PROGRAM P50_RecipeControl1
VAR
	RcpIndex	: INT;
	
	iTimerCount: INT;
	OnTimer: TON;
	OffTimerOut: BOOL;
	OnTimerOut: BOOL;
	timeTrigOn: R_TRIG;
	
	bTrigOn: BOOL;
	ReverseSignal: BOOL;
	OffTimer: TOF;
	fb_RecipeSequencer : FB_RecipeSequencer;
END_VAR

IF RCP.bRcpInit THEN
	(* reset the init flag *)
	iTimerCount := 0;
	RcpIndex := 1;
	RCP.bRcpInit := FALSE;
END_IF

IF RcpIndex <= RCP.iRcpTotalStep THEN
	OnTimer(IN:=OffTimerOut, Pt:= INT_TO_TIME(500), Q=>OnTimerOut, ET=>);
	timeTrigOn(clk:=OnTimerout, Q=>bTrigOn);
	IF (bTrigOn AND RCP.iRcpOperationState) THEN
		iTimerCount := iTimerCount +1;
		bTrigOn := FALSE;
		
		IF iTimerCount <= RCP.aRecipe[RcpIndex].iRecipe[2] THEN
			fb_RecipeSequencer(nRcpIndex:=RcpIndex);
			
		ELSIF iTimerCount > RCP.aRecipe[RcpIndex].iRecipe[2] + RCP.aRecipe[RcpIndex].iRecipe[3] THEN
			iTimerCount := 0;
			RcpIndex := RcpIndex + 1;
		END_IF
	END_IF
	IF OnTimerOut = TRUE THEN
		ReverseSignal := FALSE;
	ELSE
		ReverseSignal := TRUE;
	END_IF

	OffTimer(in:=ReverseSignal, pt:= INT_TO_TIME(500), q=>OffTimerOut,et=>);
END_IF

END_PROGRAM

(* stored: Version 1.1.0.1, ProductVersion 3.1.4026.8
   POU backup1: Id {87e0b33e-d0bf-4c9c-8bf0-f839cc997cdc}, SpecialFunc None *)
